FUNCTION_BLOCK EL1862
VAR
	_io : EL1xx9_Data;
	{attribute addProperty Name "WcState"}
	_wcState : WcStateInputToggle;
	{attribute addProperty Name "Info data"}
	_infoData : InfoDataBase;
END_VAR

PROPERTY IO : REFERENCE TO EL1xx9_Data
GET
IO REF= _io;
END_GET
END_PROPERTY

PROPERTY WcState : REFERENCE TO WcStateInputToggle
GET
WcState REF= _wcState;
END_GET
END_PROPERTY

END_FUNCTION_BLOCK

(* stored: Version 1.1.0.1, ProductVersion 3.1.4024.9
   POU EL1862: Id {07847a8a-ac33-0aeb-0b48-bb6a5b8a6157}, SpecialFunc None
   Property IO: Id {1d234ff4-a142-05ae-1c4d-e3d3e7734dbd}
   Get Get: Id {6c9b3ea3-a6df-0129-1613-f096dc23fc46}
   Property WcState: Id {25124bc4-4ae9-0229-1872-55585f189537}
   Get Get: Id {33cf9120-3152-0219-21e5-e73b515acf85} *)
